{attribute addProperty BoxType "AMP8000-0030-0103-0103"}
{attribute addProperty Id "Std_InputBIT10.1251Std_InputBIT10.1252Std_InputBIT10.1253Std_InputBIT10.1254Std_InputBIT10.1255Std_InputBIT10.1256Std_InputBIT10.1257Std_InputBIT10.1258"}
{attribute addProperty CRC "2211339070"}
{attribute addProperty SizeInBites "8"}
{attribute addProperty SizeInBytes "1"}
TYPE FSOE_83CE5B3E :
STRUCT
	{attribute addProperty Name "Std_Input"}
	Std_Input : BIT;
	{attribute addProperty Name "Std_Input"}
	Std_Input_1 : BIT;
	{attribute addProperty Name "Std_Input"}
	Std_Input_2 : BIT;
	{attribute addProperty Name "Std_Input"}
	Std_Input_3 : BIT;
	{attribute addProperty Name "Std_Input"}
	Std_Input_4 : BIT;
	{attribute addProperty Name "Std_Input"}
	Std_Input_5 : BIT;
	{attribute addProperty Name "Std_Input"}
	Std_Input_6 : BIT;
	{attribute addProperty Name "Std_Input"}
	Std_Input_7 : BIT;
END_STRUCT
END_TYPE

(* stored: Version 1.2.0.0, ProductVersion 3.1.4024.9
   DUT FSOE_83CE5B3E: Id {2f8a5f80-8786-4739-95a1-01e41628228d} *)
